TYPE PuckData :
STRUCT
	RFID: DINT;
	Status: cPuckStatusEval;
	Device: DeviceData;
	PuckOnlyRoute: STRING(30);
	Side: STRING(30);
	IsCleaningEligible: BOOL;
END_STRUCT
END_TYPE

(* stored: Version 1.1.0.1, ProductVersion 3.1.4024.6
   DUT PuckData: Id {388ad6f4-fb23-41bc-81ed-df757c268418} *)
